RoboDK station: kr30 cnc 071219 julian curve 2.rdk

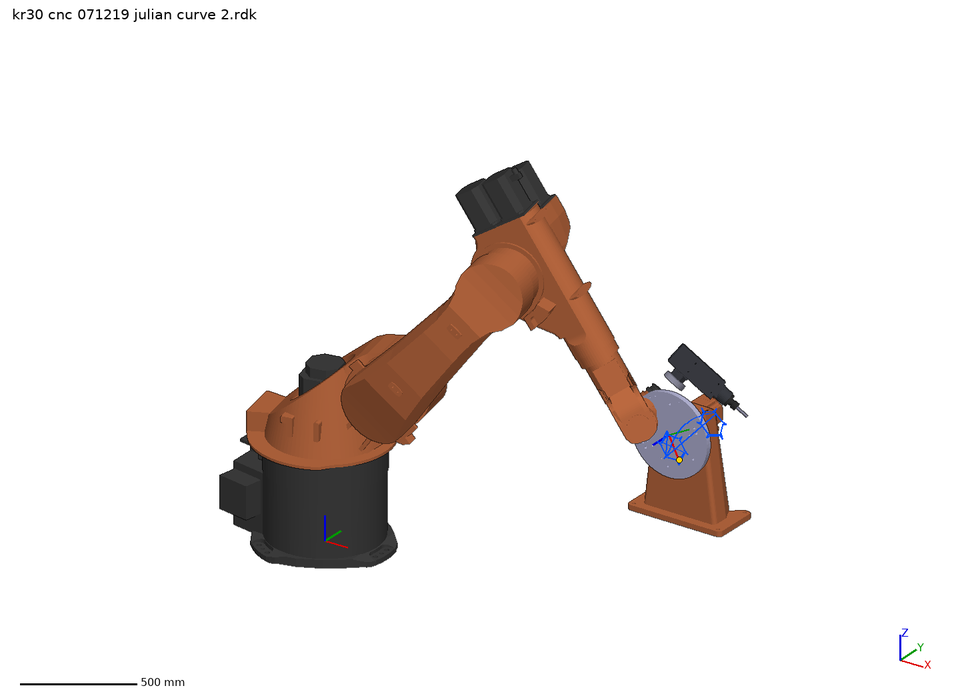
[picture v0: the station drawn from its stored meshes, robots at their saved joint values, targets as dots, program paths as lines]
Station kr30 cnc 071219 julian curve 2. Poses are relative to the parent item; angles as X-Y-Z fixed-axis rotations.
  - machining project Curve settings: C:/Temp/temp3/RhinoProject.stl | rotZ(0) | rotX(0)*rotY(0) | rotz(0) | onStart | onPathStart | onApproach | onPoint | onRetract | onFinish | onPathFinish | M_RunCode(%1)
  - frame KUKA KP1 MD250 Base at (0, 0, 0) mm
    - robot GIGASHEEN TURNTABLE OF DEATH: 1 axes, payload 250 kg
        modified DH rows (alpha deg, a mm, theta deg, d mm): 0, 0, 0, 0
        base shift (1587.22, 296.05, 828) mm, rotated rx 0 ry 90 rz -90 deg
        joint limits [-3600] to [3600]; home [0]; saved at [-332.14]
      - frame Reference Rhino at (0, 0, 0) mm
        - object RhinoPart at (0, -260, 100) mm, 30 curves
  - frame KUKA KR 30 HA Base at (0, 0, 0) mm
    - robot KUKA KR 30 HA: 6 axes, payload 30 kg, reach 2033 mm, repeatability 0.05 mm, weight 665 kg
        modified DH rows (alpha deg, a mm, theta deg, d mm): 0, 0, 0, 815; -90, 350, 0, 0; 0, 850, -90, 0; -90, 145, 0, 820; 90, 0, 0, 0; -90, 0, 180, 170
        joint limits [-185, -135, -120, -350, -119, -350] to [185, 35, 158, 350, 119, 350]; home [0, -90, 90, 0, 0, 0]; saved at [-11.373, -50.021, 107.833, -147.844, 108.332, -176.467]
      - tool 1/2" End Mill TCP, TCP at (337.71, -2.2, 160.57) mm, rotated rx 0 ry 90 rz 0 deg, size 415.8 x 102 x 153.6 mm
  - machining project RhinoPart Settings: rotZ(0) | rotX(90)*rotY(-155) | rotz(0) | onStart | onPathStart | onApproach | onPoint | onRetract | onFinish | onPathFinish | M_RunCode(%1)
  - program RhinoPart (292 instructions, listed below)
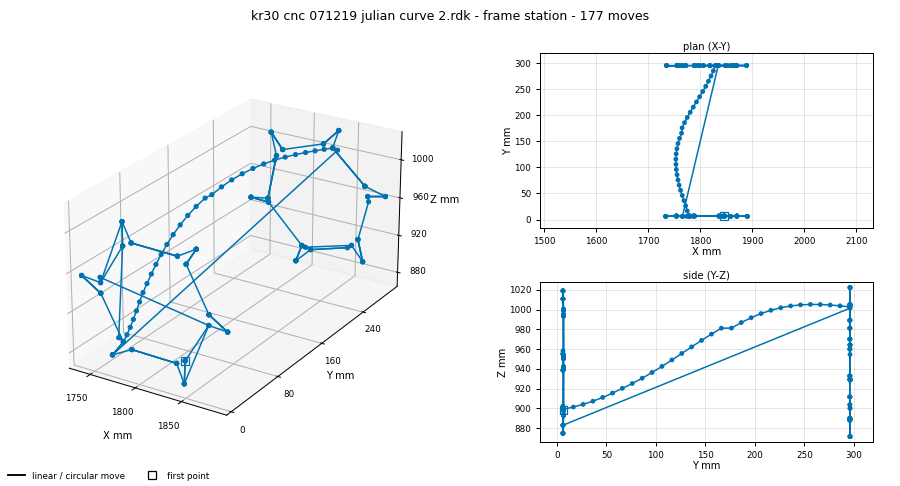
[picture p0: tool path of kr30 cnc 071219 julian curve 2.rdk in frame station, 177 of 177 moves have a stored position in this frame; points joined in program order, loops and branches not executed]

--- program RhinoPart (robot KUKA KR 30 HA) ---
  Set Ref.: Reference Rhino
  Set Tool: 1/2" End Mill TCP
  Show 1/2" End Mill TCP
  Set speed (1000.0 mm/s)
  MoveJ 1 to (58.57, 260.79, 289.44) mm, rotated rx -90 ry -25 rz -24 deg; joints [6.583, -8.141, 10.028, -24.005, 109.156, -1.613, -175.998]
  MoveL 2 to (58.57, 260.79, 289.44) mm, rotated rx -90 ry -25 rz -24 deg; joints [6.583, -8.141, 10.028, -24.005, 109.156, -1.613, -175.998]
  MoveL 3 to (58.57, 260.79, 289.44) mm, rotated rx -90 ry -25 rz -24 deg; joints [6.583, -8.141, 10.028, -24.005, 109.156, -1.613, -175.998]
  Set speed (60.0 mm/s)
  MoveL 4 to (33.55, 302.7, 289.51) mm, rotated rx -90 ry -25 rz 27.31 deg; joints [6.583, -7.995, 10.028, -23.985, 109.023, -1.55, -227.315]
  Set speed (1000.0 mm/s)
  MoveL 5 to (33.55, 302.7, 289.51) mm, rotated rx -90 ry -25 rz 27.31 deg; joints [6.583, -7.995, 10.028, -23.985, 109.023, -1.55, -227.315]
  Set speed (1000.0 mm/s)
  MoveL 6 to (-37.11, 208.63, 290) mm, rotated rx -90 ry -25 rz -135.84 deg; joints [6.7, -2.705, -6.447, -25.317, 110.179, -2.061, -54.156]
  MoveL 7 to (-32.2, 206.07, 289.37) mm, rotated rx -90 ry -25 rz -145.84 deg; joints [6.583, -8.285, 10.028, -24.026, 109.288, -1.675, -54.156]
  Set speed (60.0 mm/s)
  MoveL 8 to (-57.65, 248.19, 289.43) mm, rotated rx -90 ry -25 rz 166.78 deg; joints [6.583, -8.15, 10.028, -24.007, 109.164, -1.617, -6.784]
  Set speed (1000.0 mm/s)
  MoveL 9 to (-57.65, 248.19, 289.43) mm, rotated rx -90 ry -25 rz 166.78 deg; joints [6.583, -8.15, 10.028, -24.007, 109.164, -1.617, -6.784]
  Set speed (1000.0 mm/s)
  MoveL 10 to (21.11, 199.39, 290) mm, rotated rx -90 ry -25 rz -80.79 deg; joints [6.7, -19.001, 26.431, -23.763, 95.076, 4.976, -109.206]
  MoveL 11 to (26.13, 202.01, 289.35) mm, rotated rx -90 ry -25 rz -90.79 deg; joints [6.583, -8.312, 10.028, -24.03, 109.313, -1.687, -109.206]
  Set speed (60.0 mm/s)
  MoveL 12 to (34.79, 183.72, 290) mm, rotated rx -90 ry -25 rz -75.49 deg; joints [6.7, -4.39, -4.436, -25.266, 109.884, -1.913, -114.515]
  Set speed (1000.0 mm/s)
  MoveL 13 to (34.79, 183.72, 290) mm, rotated rx -90 ry -25 rz -75.49 deg; joints [6.7, -4.39, -4.436, -25.266, 109.884, -1.913, -114.515]
  Set speed (1000.0 mm/s)
  MoveL 14 to (26.13, 202.01, 289.35) mm, rotated rx -90 ry -25 rz -90.79 deg; joints [6.583, -8.312, 10.028, -24.03, 109.313, -1.687, -109.206]
  MoveL 15 to (26.13, 202.01, 289.35) mm, rotated rx -90 ry -25 rz -90.79 deg; joints [6.583, -8.312, 10.028, -24.03, 109.313, -1.687, -109.206]
  Set speed (60.0 mm/s)
  MoveL 16 to (-22.87, 200.95, 289.36) mm, rotated rx -90 ry -25 rz -136.21 deg; joints [6.583, -8.302, 10.028, -24.028, 109.304, -1.682, -63.793]
  Set speed (1000.0 mm/s)
  MoveL 17 to (-22.87, 200.95, 289.36) mm, rotated rx -90 ry -25 rz -136.21 deg; joints [6.583, -8.302, 10.028, -24.028, 109.304, -1.682, -63.793]
  Set speed (1000.0 mm/s)
  MoveL 18 to (-43.85, 188.95, 290) mm, rotated rx -90 ry -25 rz -131.68 deg; joints [6.7, -4.36, -4.473, -25.267, 109.891, -1.916, -58.321]
  MoveL 19 to (-43.85, 188.95, 290) mm, rotated rx -90 ry -25 rz -131.68 deg; joints [6.7, -4.36, -4.473, -25.267, 109.891, -1.916, -58.321]
  Set speed (60.0 mm/s)
  MoveL 20 to (-22.87, 200.95, 289.36) mm, rotated rx -90 ry -25 rz -136.21 deg; joints [6.583, -8.302, 10.028, -24.028, 109.304, -1.682, -63.793]
  Set speed (1000.0 mm/s)
  MoveL 21 to (-22.87, 200.95, 289.36) mm, rotated rx -90 ry -25 rz -136.21 deg; joints [6.583, -8.302, 10.028, -24.028, 109.304, -1.682, -63.793]
  Set speed (1000.0 mm/s)
  MoveL 22 to (-43.85, 188.95, 290) mm, rotated rx -90 ry -25 rz -131.68 deg; joints [6.7, -4.36, -4.473, -25.267, 109.891, -1.916, -58.321]
  MoveL 23 to (-43.85, 188.95, 290) mm, rotated rx -90 ry -25 rz -131.68 deg; joints [6.7, -4.36, -4.473, -25.267, 109.891, -1.916, -58.321]
  Set speed (60.0 mm/s)
  MoveL 24 to (-32.2, 206.07, 289.37) mm, rotated rx -90 ry -25 rz -145.84 deg; joints [6.583, -8.285, 10.028, -24.026, 109.288, -1.675, -54.156]
  Set speed (1000.0 mm/s)
  MoveL 25 to (-32.2, 206.07, 289.37) mm, rotated rx -90 ry -25 rz -145.84 deg; joints [6.583, -8.285, 10.028, -24.026, 109.288, -1.675, -54.156]
  Set speed (1000.0 mm/s)
  MoveL 26 to (-78.63, 259.66, 290) mm, rotated rx -90 ry -25 rz 170.25 deg; joints [6.7, -18.801, 25.04, -23.81, 96.165, 4.494, -0.245]
  MoveL 27 to (-78.63, 259.66, 290) mm, rotated rx -90 ry -25 rz 170.25 deg; joints [6.7, -18.801, 25.04, -23.81, 96.165, 4.494, -0.245]
  Set speed (60.0 mm/s)
  MoveL 28 to (-57.65, 248.19, 289.43) mm, rotated rx -90 ry -25 rz 166.78 deg; joints [6.583, -8.15, 10.028, -24.007, 109.164, -1.617, -6.784]
  Set speed (1000.0 mm/s)
  MoveL 29 to (-57.65, 248.19, 289.43) mm, rotated rx -90 ry -25 rz 166.78 deg; joints [6.583, -8.15, 10.028, -24.007, 109.164, -1.617, -6.784]
  Set speed (1000.0 mm/s)
  MoveL 30 to (-78.63, 259.66, 290) mm, rotated rx -90 ry -25 rz 170.25 deg; joints [6.7, -18.801, 25.04, -23.81, 96.165, 4.494, -0.245]
  MoveL 31 to (-78.63, 259.66, 290) mm, rotated rx -90 ry -25 rz 170.25 deg; joints [6.7, -18.801, 25.04, -23.81, 96.165, 4.494, -0.245]
  Set speed (60.0 mm/s)
  MoveL 32 to (-57.84, 258.86, 289.45) mm, rotated rx -90 ry -25 rz 156.39 deg; joints [6.583, -8.116, 10.028, -24.002, 109.133, -1.602, 3.606]
  Set speed (1000.0 mm/s)
  MoveL 33 to (-57.84, 258.86, 289.45) mm, rotated rx -90 ry -25 rz 156.39 deg; joints [6.583, -8.116, 10.028, -24.002, 109.133, -1.602, 3.606]
  Set speed (1000.0 mm/s)
  MoveL 34 to (-33.86, 301.87, 289.51) mm, rotated rx -90 ry -25 rz 104.47 deg; joints [6.583, -7.979, 10.028, -23.983, 109.009, -1.543, 55.533]
  MoveL 35 to (-33.86, 301.87, 289.51) mm, rotated rx -90 ry -25 rz 104.47 deg; joints [6.583, -7.979, 10.028, -23.983, 109.009, -1.543, 55.533]
  Set speed (60.0 mm/s)
  MoveL 36 to (-57.84, 258.86, 289.45) mm, rotated rx -90 ry -25 rz 156.39 deg; joints [6.583, -8.116, 10.028, -24.002, 109.133, -1.602, 3.606]
  Set speed (1000.0 mm/s)
  MoveL 37 to (-57.84, 258.86, 289.45) mm, rotated rx -90 ry -25 rz 156.39 deg; joints [6.583, -8.116, 10.028, -24.002, 109.133, -1.602, 3.606]
  Set speed (1000.0 mm/s)
  MoveL 38 to (-33.86, 301.87, 289.51) mm, rotated rx -90 ry -25 rz 104.47 deg; joints [6.583, -7.979, 10.028, -23.983, 109.009, -1.543, 55.533]
  MoveL 39 to (-33.86, 301.87, 289.51) mm, rotated rx -90 ry -25 rz 104.47 deg; joints [6.583, -7.979, 10.028, -23.983, 109.009, -1.543, 55.533]
  Set speed (60.0 mm/s)
  MoveL 40 to (-34.79, 325.15, 290) mm, rotated rx -90 ry -25 rz 108.1 deg; joints [6.7, -3.545, -5.465, -25.294, 110.05, -1.996, 61.899]
  Set speed (1000.0 mm/s)
  MoveL 41 to (-34.79, 325.15, 290) mm, rotated rx -90 ry -25 rz 108.1 deg; joints [6.7, -3.545, -5.465, -25.294, 110.05, -1.996, 61.899]
  Set speed (1000.0 mm/s)
  MoveL 42 to (-24.7, 307.31, 289.52) mm, rotated rx -90 ry -25 rz 93.11 deg; joints [6.583, -7.963, 10.028, -23.98, 108.994, -1.536, 66.89]
  MoveL 43 to (-24.7, 307.31, 289.52) mm, rotated rx -90 ry -25 rz 93.11 deg; joints [6.583, -7.963, 10.028, -23.98, 108.994, -1.536, 66.89]
  Set speed (60.0 mm/s)
  MoveL 44 to (-34.79, 325.15, 290) mm, rotated rx -90 ry -25 rz 108.1 deg; joints [6.7, -3.545, -5.465, -25.294, 110.05, -1.996, 61.899]
  Set speed (1000.0 mm/s)
  MoveL 45 to (-34.79, 325.15, 290) mm, rotated rx -90 ry -25 rz 108.1 deg; joints [6.7, -3.545, -5.465, -25.294, 110.05, -1.996, 61.899]
  Set speed (1000.0 mm/s)
  MoveL 46 to (-24.7, 307.31, 289.52) mm, rotated rx -90 ry -25 rz 93.11 deg; joints [6.583, -7.963, 10.028, -23.98, 108.994, -1.536, 66.89]
  MoveL 47 to (-24.7, 307.31, 289.52) mm, rotated rx -90 ry -25 rz 93.11 deg; joints [6.583, -7.963, 10.028, -23.98, 108.994, -1.536, 66.89]
  Set speed (60.0 mm/s)
  MoveL 48 to (24.32, 307.88, 289.52) mm, rotated rx -90 ry -25 rz 38.58 deg; joints [6.583, -7.974, 10.028, -23.982, 109.004, -1.541, 121.418]
  Set speed (1000.0 mm/s)
  MoveL 49 to (24.32, 307.88, 289.52) mm, rotated rx -90 ry -25 rz 38.58 deg; joints [6.583, -7.974, 10.028, -23.982, 109.004, -1.541, 121.418]
  Set speed (1000.0 mm/s)
  MoveL 50 to (43.85, 319.91, 290) mm, rotated rx -90 ry -25 rz 43.8 deg; joints [6.7, -3.577, -5.426, -25.293, 110.045, -1.993, 126.197]
  MoveL 51 to (43.85, 319.91, 290) mm, rotated rx -90 ry -25 rz 43.8 deg; joints [6.7, -3.577, -5.426, -25.293, 110.045, -1.993, 126.197]
  Set speed (60.0 mm/s)
  MoveL 52 to (24.32, 307.88, 289.52) mm, rotated rx -90 ry -25 rz 38.58 deg; joints [6.583, -7.974, 10.028, -23.982, 109.004, -1.541, 121.418]
  Set speed (1000.0 mm/s)
  MoveL 53 to (24.32, 307.88, 289.52) mm, rotated rx -90 ry -25 rz 38.58 deg; joints [6.583, -7.974, 10.028, -23.982, 109.004, -1.541, 121.418]
  Set speed (1000.0 mm/s)
  MoveL 54 to (43.85, 319.91, 290) mm, rotated rx -90 ry -25 rz 43.8 deg; joints [6.7, -3.577, -5.426, -25.293, 110.045, -1.993, 126.197]
  MoveL 55 to (43.85, 319.91, 290) mm, rotated rx -90 ry -25 rz 43.8 deg; joints [6.7, -3.577, -5.426, -25.293, 110.045, -1.993, 126.197]
  Set speed (60.0 mm/s)
  MoveL 56 to (33.55, 302.7, 289.51) mm, rotated rx -90 ry -25 rz 27.31 deg; joints [6.583, -7.995, 10.028, -23.985, 109.023, -1.55, 132.685]
  Set speed (1000.0 mm/s)
  MoveL 57 to (33.55, 302.7, 289.51) mm, rotated rx -90 ry -25 rz 27.31 deg; joints [6.583, -7.995, 10.028, -23.985, 109.023, -1.55, 132.685]
  Set speed (1000.0 mm/s)
  MoveL 58 to (78.63, 249.2, 290) mm, rotated rx -90 ry -25 rz -17.82 deg; joints [6.7, -4.006, -4.909, -25.279, 109.964, -1.953, 187.819]
  MoveL 59 to (78.63, 249.2, 290) mm, rotated rx -90 ry -25 rz -17.82 deg; joints [6.7, -4.006, -4.909, -25.279, 109.964, -1.953, 187.819]
  Set speed (60.0 mm/s)
  MoveL 60 to (58.57, 260.79, 289.44) mm, rotated rx -90 ry -25 rz -24 deg; joints [6.583, -8.141, 10.028, -24.005, 109.156, -1.613, 184.002]
  Set speed (1000.0 mm/s)
  MoveL 61 to (58.57, 260.79, 289.44) mm, rotated rx -90 ry -25 rz -24 deg; joints [6.583, -8.141, 10.028, -24.005, 109.156, -1.613, 184.002]
  Set speed (1000.0 mm/s)
  MoveL 62 to (78.63, 249.2, 290) mm, rotated rx -90 ry -25 rz -17.82 deg; joints [6.7, -18.788, 24.964, -23.813, 96.223, 4.468, 187.819]
  MoveL 63 to (78.63, 249.2, 290) mm, rotated rx -90 ry -25 rz -17.82 deg; joints [6.7, -18.788, 24.964, -23.813, 96.223, 4.468, 187.819]
  Set speed (60.0 mm/s)
  MoveL 64 to (58.76, 250.24, 289.42) mm, rotated rx -90 ry -25 rz -34.27 deg; joints [6.583, -8.174, 10.028, -24.01, 109.187, -1.627, 194.265]
  Set speed (1000.0 mm/s)
  MoveL 65 to (58.76, 250.24, 289.42) mm, rotated rx -90 ry -25 rz -34.27 deg; joints [6.583, -8.174, 10.028, -24.01, 109.187, -1.627, 194.265]
  Set speed (1000.0 mm/s)
  MoveL 66 to (35.18, 207.5, 289.36) mm, rotated rx -90 ry -25 rz -81.2 deg; joints [6.583, -8.298, 10.028, -24.028, 109.3, -1.681, 241.204]
  MoveL 67 to (35.18, 207.5, 289.36) mm, rotated rx -90 ry -25 rz -81.2 deg; joints [6.583, -8.298, 10.028, -24.028, 109.3, -1.681, 241.204]
  Set speed (60.0 mm/s)
  MoveL 68 to (58.76, 250.24, 289.42) mm, rotated rx -90 ry -25 rz -34.27 deg; joints [6.583, -8.174, 10.028, -24.01, 109.187, -1.627, 194.265]
  Set speed (1000.0 mm/s)
  MoveL 69 to (58.76, 250.24, 289.42) mm, rotated rx -90 ry -25 rz -34.27 deg; joints [6.583, -8.174, 10.028, -24.01, 109.187, -1.627, 194.265]
  Set speed (1000.0 mm/s)
  MoveL 70 to (35.18, 207.5, 289.36) mm, rotated rx -90 ry -25 rz -81.2 deg; joints [6.583, -8.298, 10.028, -24.028, 109.3, -1.681, 241.204]
  MoveL 71 to (35.18, 207.5, 289.36) mm, rotated rx -90 ry -25 rz -81.2 deg; joints [6.583, -8.298, 10.028, -24.028, 109.3, -1.681, 241.204]
  Set speed (60.0 mm/s)
  MoveL 72 to (34.79, 183.72, 290) mm, rotated rx -90 ry -25 rz -75.49 deg; joints [6.7, -4.39, -4.436, -25.266, 109.884, -1.913, 245.485]
  Set speed (1000.0 mm/s)
  MoveL 73 to (34.79, 183.72, 290) mm, rotated rx -90 ry -25 rz -75.49 deg; joints [6.7, -4.39, -4.436, -25.266, 109.884, -1.913, 245.485]
  Set speed (1000.0 mm/s)
  MoveL 74 to (-37.62, 299.82, 0) mm, rotated rx -90 ry -25 rz 113.38 deg; joints [-1.665, -2.525, -1.147, -27.442, 110.58, -12.079, 406.623]
  MoveL 75 to (-41.31, 295.61, 0.16) mm, rotated rx -90 ry -25 rz 103.38 deg; joints [-1.646, -5.41, 10.028, -28.034, 112.099, -12.911, 406.623]
  Set speed (60.0 mm/s)
  MoveL 76 to (4.72, 313.03, 0.16) mm, rotated rx -90 ry -25 rz 49.05 deg; joints [-1.646, -5.366, 10.028, -28.025, 112.06, -12.889, 460.953]
  Set speed (1000.0 mm/s)
  MoveL 77 to (4.72, 313.03, 0.16) mm, rotated rx -90 ry -25 rz 49.05 deg; joints [-1.646, -5.366, 10.028, -28.025, 112.06, -12.889, 460.953]
  Set speed (1000.0 mm/s)
  MoveL 78 to (-41.31, 295.61, 0.16) mm, rotated rx -90 ry -25 rz 103.38 deg; joints [-1.646, -5.41, 10.028, -28.034, 112.099, -12.911, 406.623]
  MoveL 79 to (-41.31, 295.61, 0.16) mm, rotated rx -90 ry -25 rz 103.38 deg; joints [-1.646, -5.41, 10.028, -28.034, 112.099, -12.911, 406.623]
  Set speed (60.0 mm/s)
  MoveL 80 to (-55.59, 310.29, 0) mm, rotated rx -90 ry -25 rz 117.87 deg; joints [-1.665, -4.344, 1.149, -27.361, 110.156, -11.844, 402.13]
  Set speed (1000.0 mm/s)
  MoveL 81 to (-55.59, 310.29, 0) mm, rotated rx -90 ry -25 rz 117.87 deg; joints [-1.665, -4.344, 1.149, -27.361, 110.156, -11.844, 402.13]
  Set speed (1000.0 mm/s)
  MoveL 82 to (-48.05, 287.37, 0.16) mm, rotated rx -90 ry -25 rz 114.48 deg; joints [-1.646, -5.436, 10.028, -28.039, 112.122, -12.924, 395.516]
  MoveL 83 to (-48.05, 287.37, 0.16) mm, rotated rx -90 ry -25 rz 114.48 deg; joints [-1.646, -5.436, 10.028, -28.039, 112.122, -12.924, 395.516]
  Set speed (60.0 mm/s)
  MoveL 84 to (-55.59, 310.29, 0) mm, rotated rx -90 ry -25 rz 117.87 deg; joints [-1.665, -4.344, 1.149, -27.361, 110.156, -11.844, 402.13]
  Set speed (1000.0 mm/s)
  MoveL 85 to (-55.59, 310.29, 0) mm, rotated rx -90 ry -25 rz 117.87 deg; joints [-1.665, -4.344, 1.149, -27.361, 110.156, -11.844, 402.13]
  Set speed (1000.0 mm/s)
  MoveL 86 to (-48.05, 287.37, 0.16) mm, rotated rx -90 ry -25 rz 114.48 deg; joints [-1.646, -5.436, 10.028, -28.039, 112.122, -12.924, 395.516]
  MoveL 87 to (-48.05, 287.37, 0.16) mm, rotated rx -90 ry -25 rz 114.48 deg; joints [-1.646, -5.436, 10.028, -28.039, 112.122, -12.924, 395.516]
  Set speed (60.0 mm/s)
  MoveL 88 to (-55.98, 238.83, 0.17) mm, rotated rx -90 ry -25 rz 164.89 deg; joints [-1.646, -5.591, 10.028, -28.068, 112.259, -13.003, 345.106]
  Set speed (1000.0 mm/s)
  MoveL 89 to (-55.98, 238.83, 0.17) mm, rotated rx -90 ry -25 rz 164.89 deg; joints [-1.646, -5.591, 10.028, -28.068, 112.259, -13.003, 345.106]
  Set speed (1000.0 mm/s)
  MoveL 90 to (-76.17, 234.21, 0) mm, rotated rx -90 ry -25 rz 178.7 deg; joints [-1.665, -4.909, 1.919, -27.326, 109.974, -11.744, 341.297]
  MoveL 91 to (-76.17, 234.21, 0) mm, rotated rx -90 ry -25 rz 178.7 deg; joints [-1.665, -4.909, 1.919, -27.326, 109.974, -11.744, 341.297]
  Set speed (60.0 mm/s)
  MoveL 92 to (-55.98, 238.83, 0.17) mm, rotated rx -90 ry -25 rz 164.89 deg; joints [-1.646, -5.591, 10.028, -28.068, 112.259, -13.003, 345.106]
  Set speed (1000.0 mm/s)
  MoveL 93 to (-55.98, 238.83, 0.17) mm, rotated rx -90 ry -25 rz 164.89 deg; joints [-1.646, -5.591, 10.028, -28.068, 112.259, -13.003, 345.106]
  Set speed (1000.0 mm/s)
  MoveL 94 to (-76.17, 234.21, 0) mm, rotated rx -90 ry -25 rz 178.7 deg; joints [-1.665, -4.909, 1.919, -27.326, 109.974, -11.744, 341.297]
  MoveL 95 to (-76.17, 234.21, 0) mm, rotated rx -90 ry -25 rz 178.7 deg; joints [-1.665, -4.909, 1.919, -27.326, 109.974, -11.744, 341.297]
  Set speed (60.0 mm/s)
  MoveL 96 to (-52.21, 228.87, 0.18) mm, rotated rx -90 ry -25 rz 174.99 deg; joints [-1.646, -5.623, 10.028, -28.074, 112.287, -13.019, 335.014]
  Set speed (1000.0 mm/s)
  MoveL 97 to (-52.21, 228.87, 0.18) mm, rotated rx -90 ry -25 rz 174.99 deg; joints [-1.646, -5.623, 10.028, -28.074, 112.287, -13.019, 335.014]
  Set speed (1000.0 mm/s)
  MoveL 98 to (-14.15, 197.71, 0.19) mm, rotated rx -90 ry -25 rz -138.61 deg; joints [-1.646, -5.729, 10.028, -28.095, 112.38, -13.073, 288.615]
  MoveL 99 to (-14.15, 197.71, 0.19) mm, rotated rx -90 ry -25 rz -138.61 deg; joints [-1.646, -5.729, 10.028, -28.095, 112.38, -13.073, 288.615]
  Set speed (60.0 mm/s)
  MoveL 100 to (-52.21, 228.87, 0.18) mm, rotated rx -90 ry -25 rz 174.99 deg; joints [-1.646, -5.623, 10.028, -28.074, 112.287, -13.019, 335.014]
  Set speed (1000.0 mm/s)
  MoveL 101 to (-52.21, 228.87, 0.18) mm, rotated rx -90 ry -25 rz 174.99 deg; joints [-1.646, -5.623, 10.028, -28.074, 112.287, -13.019, 335.014]
  Set speed (1000.0 mm/s)
  MoveL 102 to (-14.15, 197.71, 0.19) mm, rotated rx -90 ry -25 rz -138.61 deg; joints [-1.646, -5.729, 10.028, -28.095, 112.38, -13.073, 288.615]
  MoveL 103 to (-14.15, 197.71, 0.19) mm, rotated rx -90 ry -25 rz -138.61 deg; joints [-1.646, -5.729, 10.028, -28.095, 112.38, -13.073, 288.615]
  Set speed (60.0 mm/s)
  MoveL 104 to (-20.57, 178.36, 0) mm, rotated rx -90 ry -25 rz -124.14 deg; joints [-1.665, -5.328, 2.509, -27.298, 109.822, -11.661, 284.144]
  Set speed (1000.0 mm/s)
  MoveL 105 to (-20.57, 178.36, 0) mm, rotated rx -90 ry -25 rz -124.14 deg; joints [-1.665, -5.328, 2.509, -27.298, 109.822, -11.661, 284.144]
  Set speed (1000.0 mm/s)
  MoveL 106 to (-10.16, 196.36, 0) mm, rotated rx -90 ry -25 rz -119.07 deg; joints [-1.665, -3.353, -0.136, -27.411, 110.416, -11.988, 279.071]
  MoveL 107 to (-10.16, 196.36, 0) mm, rotated rx -90 ry -25 rz -119.07 deg; joints [-1.665, -3.353, -0.136, -27.411, 110.416, -11.988, 279.071]
  Set speed (60.0 mm/s)
  MoveL 108 to (-20.57, 178.36, 0) mm, rotated rx -90 ry -25 rz -124.14 deg; joints [-1.665, -5.328, 2.509, -27.298, 109.822, -11.661, 284.144]
  Set speed (1000.0 mm/s)
  MoveL 109 to (-20.57, 178.36, 0) mm, rotated rx -90 ry -25 rz -124.14 deg; joints [-1.665, -5.328, 2.509, -27.298, 109.822, -11.661, 284.144]
  Set speed (1000.0 mm/s)
  MoveL 110 to (-10.16, 196.36, 0) mm, rotated rx -90 ry -25 rz -119.07 deg; joints [-1.665, -3.353, -0.136, -27.411, 110.416, -11.988, 279.071]
  MoveL 111 to (-10.16, 196.36, 0) mm, rotated rx -90 ry -25 rz -119.07 deg; joints [-1.665, -3.353, -0.136, -27.411, 110.416, -11.988, 279.071]
  Set speed (60.0 mm/s)
  MoveL 112 to (42.38, 213.36, 0.18) mm, rotated rx -90 ry -25 rz -83.56 deg; joints [-1.646, -5.699, 10.028, -28.089, 112.354, -13.058, 233.558]
  Set speed (1000.0 mm/s)
  MoveL 113 to (42.38, 213.36, 0.18) mm, rotated rx -90 ry -25 rz -83.56 deg; joints [-1.646, -5.699, 10.028, -28.089, 112.354, -13.058, 233.558]
  Set speed (1000.0 mm/s)
  MoveL 114 to (55.59, 198.58, 0) mm, rotated rx -90 ry -25 rz -67.85 deg; joints [-1.665, -12.832, 17.764, -26.271, 102.9, -8.022, 227.85]
  MoveL 115 to (55.59, 198.58, 0) mm, rotated rx -90 ry -25 rz -67.85 deg; joints [-1.665, -12.832, 17.764, -26.271, 102.9, -8.022, 227.85]
  Set speed (60.0 mm/s)
  MoveL 116 to (42.38, 213.36, 0.18) mm, rotated rx -90 ry -25 rz -83.56 deg; joints [-1.646, -5.699, 10.028, -28.089, 112.354, -13.058, 233.558]
  Set speed (1000.0 mm/s)
  MoveL 117 to (42.38, 213.36, 0.18) mm, rotated rx -90 ry -25 rz -83.56 deg; joints [-1.646, -5.699, 10.028, -28.089, 112.354, -13.058, 233.558]
  Set speed (1000.0 mm/s)
  MoveL 118 to (55.59, 198.58, 0) mm, rotated rx -90 ry -25 rz -67.85 deg; joints [-1.665, -12.832, 17.764, -26.271, 102.9, -8.022, 227.85]
  MoveL 119 to (55.59, 198.58, 0) mm, rotated rx -90 ry -25 rz -67.85 deg; joints [-1.665, -12.832, 17.764, -26.271, 102.9, -8.022, 227.85]
  Set speed (60.0 mm/s)
  MoveL 120 to (49.13, 221.59, 0.18) mm, rotated rx -90 ry -25 rz -73.83 deg; joints [-1.646, -5.677, 10.028, -28.085, 112.334, -13.046, 223.831]
  Set speed (1000.0 mm/s)
  MoveL 121 to (49.13, 221.59, 0.18) mm, rotated rx -90 ry -25 rz -73.83 deg; joints [-1.646, -5.677, 10.028, -28.085, 112.334, -13.046, 223.831]
  Set speed (1000.0 mm/s)
  MoveL 122 to (58.12, 264.32, 0) mm, rotated rx -90 ry -25 rz -15.75 deg; joints [-1.665, -13.53, 20.853, -26.05, 100.754, -6.946, 175.746]
  MoveL 123 to (57.11, 270.16, 0.17) mm, rotated rx -90 ry -25 rz -25.75 deg; joints [-1.646, -5.529, 10.028, -28.056, 112.203, -12.971, 175.746]
  Set speed (60.0 mm/s)
  MoveL 124 to (45.21, 216.6, 0) mm, rotated rx -90 ry -25 rz -63.83 deg; joints [-1.665, -13.449, 20.388, -26.083, 101.099, -7.117, 223.831]
  Set speed (1000.0 mm/s)
  MoveL 125 to (49.13, 221.59, 0.18) mm, rotated rx -90 ry -25 rz -73.83 deg; joints [-1.646, -5.677, 10.028, -28.085, 112.334, -13.046, 223.831]
  Set speed (1000.0 mm/s)
  MoveL 126 to (58.12, 264.32, 0) mm, rotated rx -90 ry -25 rz -15.75 deg; joints [-1.665, -13.53, 20.853, -26.05, 100.754, -6.946, 175.746]
  MoveL 127 to (57.11, 270.16, 0.17) mm, rotated rx -90 ry -25 rz -25.75 deg; joints [-1.646, -5.529, 10.028, -28.056, 112.203, -12.971, 175.746]
  Set speed (60.0 mm/s)
  MoveL 128 to (76.17, 274.65, 0) mm, rotated rx -90 ry -25 rz -9.11 deg; joints [-1.665, -4.609, 1.506, -27.345, 110.074, -11.799, 169.111]
  Set speed (1000.0 mm/s)
  MoveL 129 to (76.17, 274.65, 0) mm, rotated rx -90 ry -25 rz -9.11 deg; joints [-1.665, -4.609, 1.506, -27.345, 110.074, -11.799, 169.111]
  Set speed (1000.0 mm/s)
  MoveL 130 to (53.34, 280.13, 0.17) mm, rotated rx -90 ry -25 rz -15.16 deg; joints [-1.646, -5.495, 10.028, -28.05, 112.174, -12.954, 165.162]
  MoveL 131 to (53.34, 280.13, 0.17) mm, rotated rx -90 ry -25 rz -15.16 deg; joints [-1.646, -5.495, 10.028, -28.05, 112.174, -12.954, 165.162]
  Set speed (60.0 mm/s)
  MoveL 132 to (76.17, 274.65, 0) mm, rotated rx -90 ry -25 rz -9.11 deg; joints [-1.665, -4.609, 1.506, -27.345, 110.074, -11.799, 169.111]
  Set speed (1000.0 mm/s)
  MoveL 133 to (76.17, 274.65, 0) mm, rotated rx -90 ry -25 rz -9.11 deg; joints [-1.665, -4.609, 1.506, -27.345, 110.074, -11.799, 169.111]
  Set speed (1000.0 mm/s)
  MoveL 134 to (53.34, 280.13, 0.17) mm, rotated rx -90 ry -25 rz -15.16 deg; joints [-1.646, -5.495, 10.028, -28.05, 112.174, -12.954, 165.162]
  MoveL 135 to (53.34, 280.13, 0.17) mm, rotated rx -90 ry -25 rz -15.16 deg; joints [-1.646, -5.495, 10.028, -28.05, 112.174, -12.954, 165.162]
  Set speed (60.0 mm/s)
  MoveL 136 to (20.49, 309.71, 0) mm, rotated rx -90 ry -25 rz 47.6 deg; joints [-1.665, -2.442, -1.246, -27.445, 110.594, -12.086, 112.405]
  Set speed (1000.0 mm/s)
  MoveL 137 to (15.24, 311.32, 0.16) mm, rotated rx -90 ry -25 rz 37.6 deg; joints [-1.646, -5.376, 10.028, -28.027, 112.069, -12.894, 112.405]
  Set speed (1000.0 mm/s)
  MoveL 138 to (20.57, 330.51, 0) mm, rotated rx -90 ry -25 rz 53.73 deg; joints [-1.665, -4.194, 0.95, -27.369, 110.2, -11.868, 106.267]
  MoveL 139 to (20.57, 330.51, 0) mm, rotated rx -90 ry -25 rz 53.73 deg; joints [-1.665, -4.194, 0.95, -27.369, 110.2, -11.868, 106.267]
  Set speed (60.0 mm/s)
  MoveL 140 to (15.24, 311.32, 0.16) mm, rotated rx -90 ry -25 rz 37.6 deg; joints [-1.646, -5.376, 10.028, -28.027, 112.069, -12.894, 112.405]
  Set speed (1000.0 mm/s)
  MoveL 141 to (15.24, 311.32, 0.16) mm, rotated rx -90 ry -25 rz 37.6 deg; joints [-1.646, -5.376, 10.028, -28.027, 112.069, -12.894, 112.405]
  Set speed (1000.0 mm/s)
  MoveL 142 to (20.57, 330.51, 0) mm, rotated rx -90 ry -25 rz 53.73 deg; joints [-1.665, -13.179, 19.106, -26.174, 102.007, -7.572, 106.267]
  MoveL 143 to (20.57, 330.51, 0) mm, rotated rx -90 ry -25 rz 53.73 deg; joints [-1.665, -13.179, 19.106, -26.174, 102.007, -7.572, 106.267]
  Set speed (60.0 mm/s)
  MoveL 144 to (4.72, 313.03, 0.16) mm, rotated rx -90 ry -25 rz 49.05 deg; joints [-1.646, -5.366, 10.028, -28.025, 112.06, -12.889, 100.953]
  Set speed (1000.0 mm/s)
  MoveL 145 to (4.72, 313.03, 0.16) mm, rotated rx -90 ry -25 rz 49.05 deg; joints [-1.646, -5.366, 10.028, -28.025, 112.06, -12.889, 100.953]
  Set speed (1000.0 mm/s)
  MoveL 146 to (-41.31, 295.61, 0.16) mm, rotated rx -90 ry -25 rz 103.38 deg; joints [-1.646, -5.41, 10.028, -28.034, 112.099, -12.911, 46.623]
  MoveL 147 to (-41.31, 295.61, 0.16) mm, rotated rx -90 ry -25 rz 103.38 deg; joints [-1.646, -5.41, 10.028, -28.034, 112.099, -12.911, 46.623]
  Set speed (60.0 mm/s)
  MoveL 148 to (-44.05, 292.64, 10.13) mm, rotated rx -90 ry -25 rz 107.89 deg; joints [-1.364, -5.421, 10.028, -27.912, 112.24, -12.648, 42.114]
  MoveL 149 to (-46.87, 289.1, 20.1) mm, rotated rx -90 ry -25 rz 112.81 deg; joints [-1.082, -5.434, 10.028, -27.79, 112.383, -12.386, 37.19]
  MoveL 150 to (-49.64, 284.97, 30.07) mm, rotated rx -90 ry -25 rz 118.1 deg; joints [-0.8, -5.448, 10.028, -27.667, 112.526, -12.124, 31.9]
  MoveL 151 to (-52.22, 280.27, 40.04) mm, rotated rx -90 ry -25 rz 123.71 deg; joints [-0.518, -5.463, 10.028, -27.544, 112.67, -11.861, 26.29]
  MoveL 152 to (-54.49, 275, 50.02) mm, rotated rx -90 ry -25 rz 129.59 deg; joints [-0.235, -5.481, 10.028, -27.42, 112.816, -11.599, 20.409]
  MoveL 153 to (-56.32, 269.22, 60) mm, rotated rx -90 ry -25 rz 135.7 deg; joints [0.047, -5.499, 10.028, -27.296, 112.961, -11.337, 14.303]
  MoveL 154 to (-57.57, 262.99, 69.97) mm, rotated rx -90 ry -25 rz 141.99 deg; joints [0.329, -5.519, 10.028, -27.171, 113.108, -11.075, 8.015]
  MoveL 155 to (-58.15, 256.4, 79.94) mm, rotated rx -90 ry -25 rz 148.41 deg; joints [0.611, -5.54, 10.028, -27.045, 113.254, -10.813, 1.589]
  MoveL 156 to (-57.96, 249.58, 89.92) mm, rotated rx -90 ry -25 rz 154.94 deg; joints [0.894, -5.561, 10.028, -26.919, 113.401, -10.551, -4.936]
  MoveL 157 to (-56.94, 242.64, 99.88) mm, rotated rx -90 ry -25 rz 161.52 deg; joints [1.176, -5.582, 10.028, -26.793, 113.547, -10.287, -11.521]
  MoveL 158 to (-55.05, 235.74, 109.85) mm, rotated rx -90 ry -25 rz 168.13 deg; joints [1.458, -5.602, 10.028, -26.665, 113.692, -10.023, -18.132]
  MoveL 159 to (-52.28, 229.02, 119.81) mm, rotated rx -90 ry -25 rz 174.74 deg; joints [1.74, -5.622, 10.028, -26.537, 113.835, -9.758, -24.736]
  MoveL 160 to (-52.68, 227.97, 130) mm, rotated rx -90 ry -25 rz -168.7 deg; joints [2.045, -3.265, -0.119, -26.333, 111.997, -8.394, -31.302]
  MoveL 161 to (-49.15, 221.88, 140) mm, rotated rx -90 ry -25 rz -162.2 deg; joints [2.33, -3.459, 0.239, -26.217, 111.975, -8.041, -37.801]
  MoveL 162 to (-44.94, 216.28, 150) mm, rotated rx -90 ry -25 rz -155.79 deg; joints [2.615, -3.675, 0.646, -26.095, 111.93, -7.675, -44.207]
  MoveL 163 to (-40.17, 211.29, 160) mm, rotated rx -90 ry -25 rz -149.51 deg; joints [2.899, -3.915, 1.107, -25.968, 111.857, -7.295, -50.492]
  MoveL 164 to (-34.94, 206.95, 170) mm, rotated rx -90 ry -25 rz -143.37 deg; joints [3.184, -4.185, 1.63, -25.835, 111.752, -6.9, -56.632]
  MoveL 165 to (-29.38, 203.32, 180) mm, rotated rx -90 ry -25 rz -137.4 deg; joints [3.468, -4.488, 2.229, -25.694, 111.611, -6.487, -62.601]
  MoveL 166 to (-23.62, 200.42, 190) mm, rotated rx -90 ry -25 rz -131.63 deg; joints [3.753, -4.836, 2.92, -25.545, 111.423, -6.052, -68.373]
  MoveL 167 to (-17.8, 198.23, 200) mm, rotated rx -90 ry -25 rz -126.08 deg; joints [4.037, -5.242, 3.735, -25.385, 111.176, -5.588, -73.923]
  MoveL 168 to (-12.04, 196.73, 210) mm, rotated rx -90 ry -25 rz -120.78 deg; joints [4.321, -5.737, 4.732, -25.21, 110.843, -5.083, -79.224]
  MoveL 169 to (-6.46, 195.84, 220) mm, rotated rx -90 ry -25 rz -115.75 deg; joints [4.604, -6.386, 6.046, -25.011, 110.361, -4.507, -84.249]
  MoveL 170 to (-1.16, 195.49, 230) mm, rotated rx -90 ry -25 rz -111.03 deg; joints [4.888, -7.495, 8.294, -24.743, 109.448, -3.724, -88.971]
  MoveL 171 to (4.44, 195.74, 239.94) mm, rotated rx -90 ry -25 rz -106.64 deg; joints [5.171, -8.348, 10.028, -24.521, 108.765, -3.064, -93.359]
  MoveL 172 to (9.8, 196.5, 249.85) mm, rotated rx -90 ry -25 rz -102.62 deg; joints [5.454, -8.342, 10.028, -24.424, 108.877, -2.789, -97.383]
  MoveL 173 to (14.69, 197.62, 259.75) mm, rotated rx -90 ry -25 rz -98.99 deg; joints [5.737, -8.335, 10.028, -24.326, 108.987, -2.514, -101.013]
  MoveL 174 to (19.05, 198.99, 269.63) mm, rotated rx -90 ry -25 rz -95.79 deg; joints [6.019, -8.328, 10.028, -24.228, 109.097, -2.238, -104.215]
  MoveL 175 to (22.87, 200.49, 279.5) mm, rotated rx -90 ry -25 rz -93.04 deg; joints [6.301, -8.32, 10.028, -24.129, 109.205, -1.963, -106.957]
  MoveL 176 to (26.13, 202.01, 289.35) mm, rotated rx -90 ry -25 rz -90.79 deg; joints [6.583, -8.312, 10.028, -24.03, 109.313, -1.687, -109.206]
  Set speed (1000.0 mm/s)
  MoveL 177 to (26.13, 202.01, 289.35) mm, rotated rx -90 ry -25 rz -90.79 deg; joints [6.583, -8.312, 10.028, -24.03, 109.313, -1.687, -109.206]
  Set speed (1000.0 mm/s)
